FUNCTION_BLOCK OC_DONE (* CAT Function Block Type *)
  (* Standard: 61499-2 *)
  (* Version 0.0, 7/10/2026, Schneider Electric, template *)
  PACKAGE SE.Nereda;
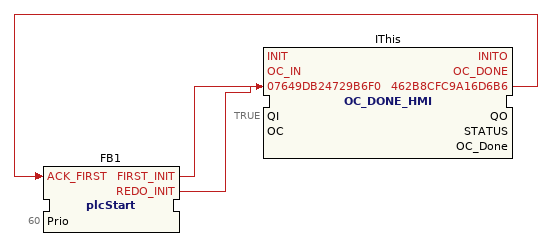
  FBS
    IThis : OC_DONE_HMI(QI := TRUE);
    FB1 : plcStart(Prio := 60);
  END_FBS
  EVENT_CONNECTIONS
    FB1.FIRST_INIT TO IThis.07649DB24729B6F0;
    FB1.REDO_INIT TO IThis.07649DB24729B6F0;
    IThis.462B8CFC9A16D6B6 TO FB1.ACK_FIRST;
  END_CONNECTIONS
END_FUNCTION_BLOCK
